(* CoDeSys 2.3.9.41 project: Собственные функциональные блоки.pro *)

(* POU PLC_PRG, CFC *)
PROGRAM PLC_PRG
VAR
	slojeniya: Arifmetika;
	in1: REAL;
	in2: REAL;
	out1: REAL;
	deleniya: Arifmetika1;
	in3: REAL;
	in4: REAL;
	out2: REAL;
	vichitanie: Arifmetika2;
	in5: REAL;
	in6: REAL;
	out3: REAL;
	umnojenie: Arifmetika3;
	in7: REAL;
	in8: REAL;
	out4: REAL;
	X: REAL;
	Xmin: REAL;
	Xmax: REAL;
	Ymin: REAL;
	Ymax: REAL;
	Y: REAL;
	masshtab: Masshtabirovanie;
END_VAR
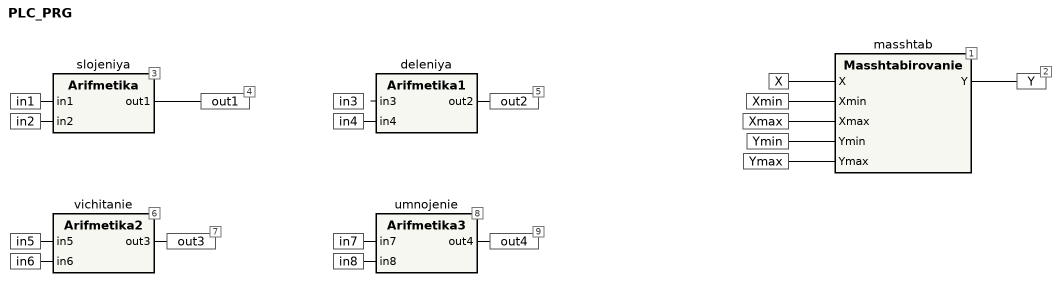
_CFC_ (* Continuous Function Chart, elements in execution order *)
unconnected input in3
#0 deleniya:Arifmetika1(in3: -, in4: in4)
#1 masshtab:Masshtabirovanie(X: X, Xmin: Xmin, Xmax: Xmax, Ymin: Ymin, Ymax: Ymax)
#2 Y <= #1.Y
#3 slojeniya:Arifmetika(in1: in1, in2: in2)
#4 out1 <= #3.out1
#5 out2 <= #0.out2
#6 vichitanie:Arifmetika2(in5: in5, in6: in6)
#7 out3 <= #6.out3
#8 umnojenie:Arifmetika3(in7: in7, in8: in8)
#9 out4 <= #8.out4
_END_CFC_
(* the same logic as Structured Text *)
deleniya(in4 := in4);
masshtab(X := X, Xmin := Xmin, Xmax := Xmax, Ymin := Ymin, Ymax := Ymax);
Y := masshtab.Y;
slojeniya(in1 := in1, in2 := in2);
out1 := slojeniya.out1;
out2 := deleniya.out2;
vichitanie(in5 := in5, in6 := in6);
out3 := vichitanie.out3;
umnojenie(in7 := in7, in8 := in8);
out4 := umnojenie.out4;
END_PROGRAM

(* POU Arifmetika, ST *)
FUNCTION_BLOCK Arifmetika
VAR_INPUT
	in1,in2:REAL;
END_VAR
VAR_OUTPUT
	out1:REAL;
END_VAR
VAR
END_VAR
out1:=in1+in2;
END_FUNCTION_BLOCK

(* POU Arifmetika1, ST *)
FUNCTION_BLOCK Arifmetika1
VAR_INPUT
	in3,in4:REAL;
END_VAR
VAR_OUTPUT
	out2:REAL;
END_VAR
VAR
END_VAR
out2:=in3/in4;
END_FUNCTION_BLOCK

(* POU Arifmetika2, ST *)
FUNCTION_BLOCK Arifmetika2
VAR_INPUT
	in5,in6:REAL;
END_VAR
VAR_OUTPUT
	out3:REAL;
END_VAR
VAR
END_VAR
out3:=in5-in6;
END_FUNCTION_BLOCK

(* POU Arifmetika3, ST *)
FUNCTION_BLOCK Arifmetika3
VAR_INPUT
	in7,in8:REAL;
END_VAR
VAR_OUTPUT
	out4:REAL;
END_VAR
VAR
END_VAR
out4:=in7*in8;
END_FUNCTION_BLOCK

(* POU Masshtabirovanie, ST *)
FUNCTION_BLOCK Masshtabirovanie
VAR_INPUT
	X:REAL;
	Xmin:REAL;
	Xmax:REAL;
	Ymin:REAL;
	Ymax:REAL;
END_VAR
VAR_OUTPUT
	Y:REAL;
END_VAR
VAR
END_VAR
IF(Xmax<>Xmin)
THEN
Y:=(Ymax-Ymin)*((X-Xmin)/(Xmax-Xmin))+Ymin;
ELSE
Y:=0.0;
END_IF
END_FUNCTION_BLOCK
